Staubli VAL3: test_ventouse.dtx

mdesc mNomSpeed = {vel=300, blend=off}
jointRx jP1
jointRx jP2 = {j1=67.72, j2=50.87, j3=100.24, j5=28.89, j6=-112.28}
jointRx jP3 = {j1=-83.94, j2=66.93, j3=62.59, j5=50.48, j6=-263.94}
tool ventouse = {z=50, fatherId=flange[0], ioLink=valve1, ioOpen=1, ioClose=1}
jointRx jP4 = {j1=67.72, j2=17.89, j3=90, j5=72.11, j6=-112.28}
jointRx jP5 = {j1=-84.94, j2=43.97, j3=50.35, j5=58.68, j6=-263.94}
public sio siSocketTCP = {link=Socket\siSocketTCP}
bool bOverRun
public sio siSocketUDP = {link=UdpSocket\siSocketUDP}
public dio doValve1 = {link=valve1}
